TYPE Pascal :
STRUCT
    _ : REAL;
END_STRUCT
END_TYPE

(* stored: Version 1.1.0.1, ProductVersion 3.1.4024.4
   DUT Pascal: Id {2022ed1b-2512-429e-89ad-9be1a2114fdc} *)
